PROGRAM MAIN
VAR
	
END_VAR

P_Task1();
P_task2();

END_PROGRAM

(* stored: Version 1.1.0.1, ProductVersion 3.1.4024.12
   POU MAIN: Id {7bc75ca4-379a-4c00-abfc-71f15484895c}, SpecialFunc None *)
